// Mitsubishi GX Works2 project: 서보, 시퀀스 회로 예시   PLC: Q03UDV

PROGRAM MAIN
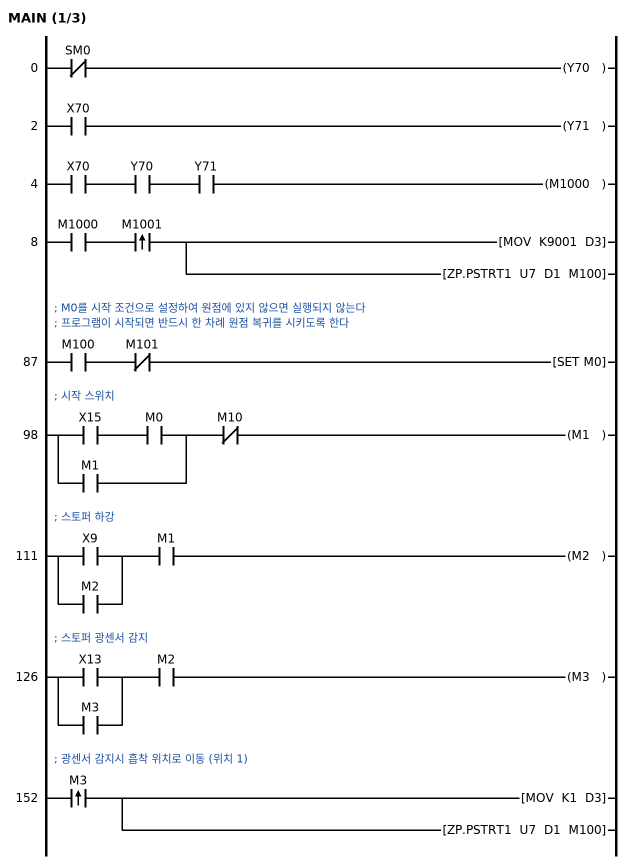
0     LDI     SM0
      OUT     Y70
2     LD      X70
      OUT     Y71
4     LD      X70
      AND     Y70
      AND     Y71
      OUT     M1000
8     LD      M1000
      ANDP    M1001
      MOV     K9001 D3
      ZP.PSTRT1 U7 D1 M100
; M0를 시작 조건으로 설정하여 원점에 있지 않으면 실행되지 않는다
; 프로그램이 시작되면 반드시 한 차례 원점 복귀를 시키도록 한다
87    LD      M100
      ANI     M101
      SET     M0
; 시작 스위치
98    LD      X15
      AND     M0
      OR      M1
      ANI     M10
      OUT     M1
; 스토퍼 하강
111   LD      X9
      OR      M2
      AND     M1
      OUT     M2
; 스토퍼 광센서 감지
126   LD      X13
      OR      M3
      AND     M2
      OUT     M3
; 광센서 감지시 흡착 위치로 이동 (위치 1)
152   LDP     M3
      MOV     K1 D3
      ZP.PSTRT1 U7 D1 M100
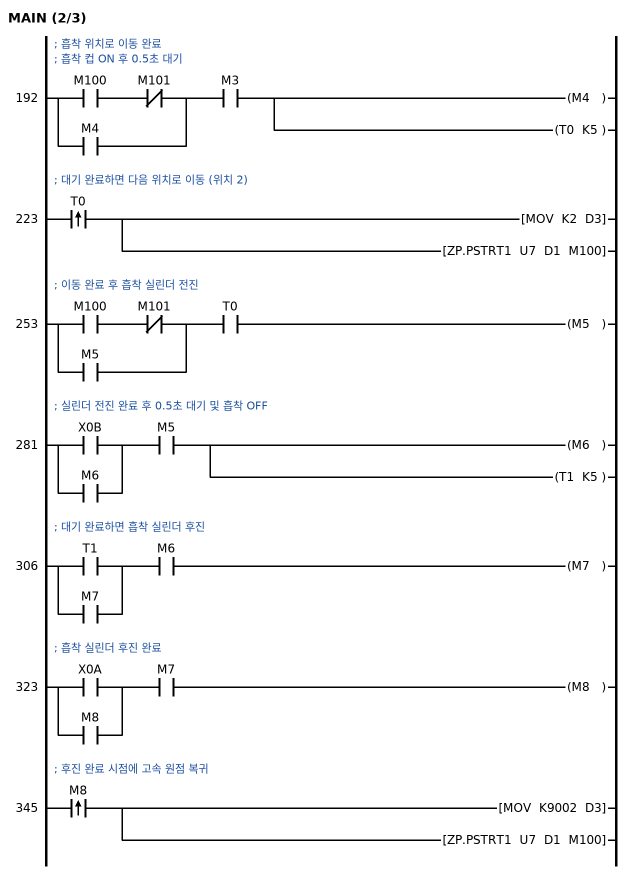
; 흡착 위치로 이동 완료
; 흡착 컵 ON 후 0.5초 대기
192   LD      M100
      ANI     M101
      OR      M4
      AND     M3
      OUT     M4
      OUT     T0 K5
; 대기 완료하면 다음 위치로 이동 (위치 2)
223   LDP     T0
      MOV     K2 D3
      ZP.PSTRT1 U7 D1 M100
; 이동 완료 후 흡착 실린더 전진
253   LD      M100
      ANI     M101
      OR      M5
      AND     T0
      OUT     M5
; 실린더 전진 완료 후 0.5초 대기 및 흡착 OFF
281   LD      X0B
      OR      M6
      AND     M5
      OUT     M6
      OUT     T1 K5
; 대기 완료하면 흡착 실린더 후진
306   LD      T1
      OR      M7
      AND     M6
      OUT     M7
; 흡착 실린더 후진 완료
323   LD      X0A
      OR      M8
      AND     M7
      OUT     M8
; 후진 완료 시점에 고속 원점 복귀
345   LDP     M8
      MOV     K9002 D3
      ZP.PSTRT1 U7 D1 M100
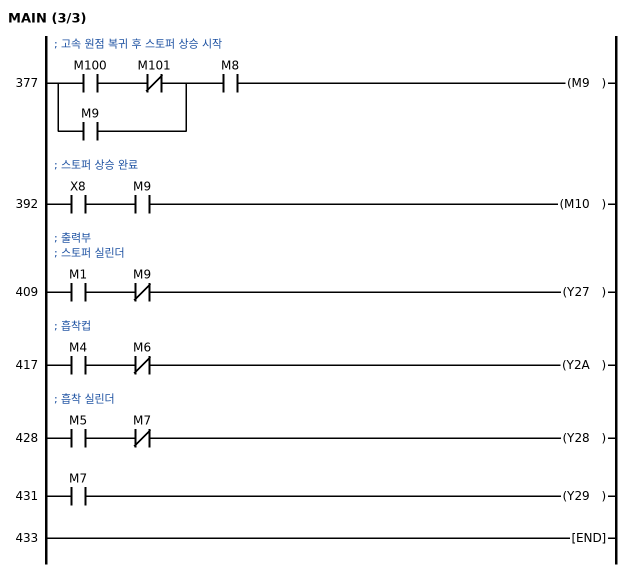
; 고속 원점 복귀 후 스토퍼 상승 시작
377   LD      M100
      ANI     M101
      OR      M9
      AND     M8
      OUT     M9
; 스토퍼 상승 완료
392   LD      X8
      AND     M9
      OUT     M10
; 출력부
; 스토퍼 실린더
409   LD      M1
      ANI     M9
      OUT     Y27
; 흡착컵
417   LD      M4
      ANI     M6
      OUT     Y2A
; 흡착 실린더
428   LD      M5
      ANI     M7
      OUT     Y28
431   LD      M7
      OUT     Y29
433   END
END_PROGRAM
